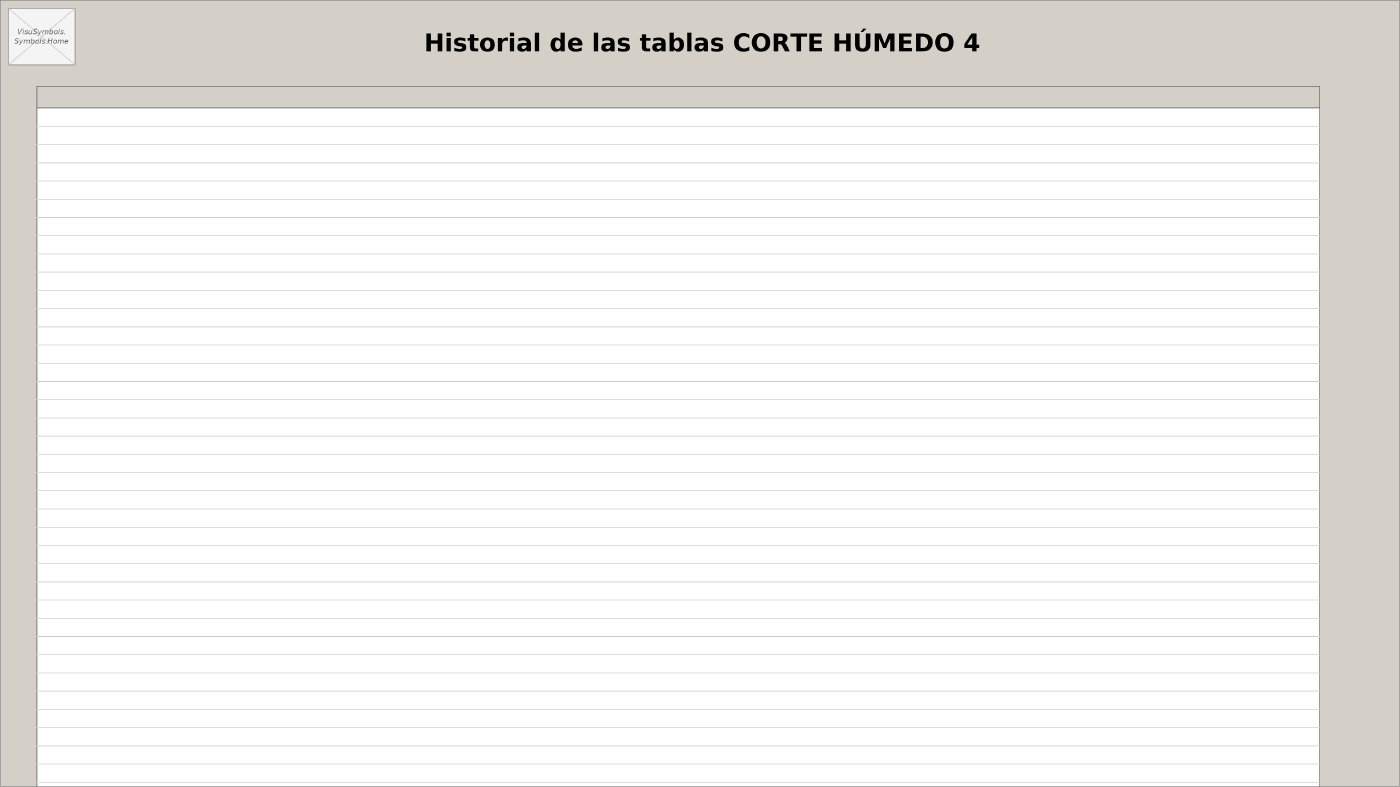
VISUALIZATION HistTablaTablas_Ch4  // 1920x1080
    Label (439,29 1048x59), "Historial de las tablas CORTE HÚMEDO 4"
    Image (11,11 92x78), image: VisuSymbols.Symbols.Home
        OnMouseClick: change screen: Home_CortH4
    Table (50,118 1760x963), data array: RegistroLocalDataBase.aHistoricStrTablasCH4
        p3854506369: RegistroLocalDataBase.aHistoricStrTablasCH4[INDEX].ID
        p1892666644: RegistroLocalDataBase.aHistoricStrTablasCH4[INDEX].Fecha
        p338671338: RegistroLocalDataBase.aHistoricStrTablasCH4[INDEX].Modelo
        p2170511999: RegistroLocalDataBase.aHistoricStrTablasCH4[INDEX].Formato
        p3723444502: RegistroLocalDataBase.aHistoricStrTablasCH4[INDEX].Espesor
        p1218418051: RegistroLocalDataBase.aHistoricStrTablasCH4[INDEX].Maquina
        p746581629: RegistroLocalDataBase.aHistoricStrTablasCH4[INDEX].Cont_Piezas
        p3104783080: RegistroLocalDataBase.aHistoricStrTablasCH4[INDEX].t_Entre_Piez_Ftc
        p2501879983: RegistroLocalDataBase.aHistoricStrTablasCH4[INDEX].S_Justi_Paro_Ftc
        p1757482276: Numero de tablas
        p4088588272: Tiempo entre tablas
        p2243050616: Justif paro
END_VISUALIZATION

(* stored: Version 1.1.0.1, ProductVersion 3.1.4024.12
   Visu HistTablaTablas_Ch4: Id {169d72ac-5c2b-4084-979b-fd36a443784b} *)
